Staubli VAL3: buildList.pgx

program buildList()
  local num l_nSize
  local string l_sEvent
  local num i
  local bool l_bFound
  local num l_nCount
  local string l_sEmpty
  local num j
begin
  call use:setSizeList(0,0,38,10)
  //call use:setSizeList(15,0,18,9)
  //建立对话款
  call use:listcreate("第1槽/6槽")
  //  for i=0 to 7
  //    call use:listadd(sMenu[i])
  //  endFor
 //   call use:selectNewField(nSelected,nIndex,nView)
  for i=0 to 7
    sTrsfNum[i,0]=toString("",data:pPoinTest[i].trsf.x)
    sTrsfNum[i,1]=toString("",data:pPoinTest[i].trsf.y)
    sTrsfNum[i,2]=toString("",data:pPoinTest[i].trsf.z)
    sTrsfNum[i,3]=toString("",data:pPoinTest[i].trsf.rx)
    sTrsfNum[i,4]=toString("",data:pPoinTest[i].trsf.ry)
    sTrsfNum[i,5]=toString("",data:pPoinTest[i].trsf.rz)
  endFor

  sWorkingmode[0]="0 安全过度点 Joint"
  sWorkingmode[1]="1 Appro(摆正点，{"+sTrsfNum[1,0]+","+sTrsfNum[1,1]+","+sTrsfNum[1,2]+","+sTrsfNum[1,3]+","+sTrsfNum[1,4]+","+sTrsfNum[1,5]+"})"
  sWorkingmode[2]="2 Appro(摆正点，{"+sTrsfNum[2,0]+","+sTrsfNum[2,1]+","+sTrsfNum[2,2]+","+sTrsfNum[2,3]+","+sTrsfNum[2,4]+","+sTrsfNum[2,5]+"})"
  sWorkingmode[3]="3 Appro(到位点，{"+sTrsfNum[3,0]+","+sTrsfNum[3,1]+","+sTrsfNum[3,2]+","+sTrsfNum[3,3]+","+sTrsfNum[3,4]+","+sTrsfNum[3,5]+"})"
  sWorkingmode[4]="4 Appro(到位点，{"+sTrsfNum[4,0]+","+sTrsfNum[4,1]+","+sTrsfNum[4,2]+","+sTrsfNum[4,3]+","+sTrsfNum[4,4]+","+sTrsfNum[4,5]+"})"
  sWorkingmode[5]="5 Appro(到位点，{"+sTrsfNum[5,0]+","+sTrsfNum[5,1]+","+sTrsfNum[5,2]+","+sTrsfNum[5,3]+","+sTrsfNum[5,4]+","+sTrsfNum[5,5]+"})"
  sWorkingmode[6]="6 Appro(摆正点，{"+sTrsfNum[6,0]+","+sTrsfNum[6,1]+","+sTrsfNum[6,2]+","+sTrsfNum[6,3]+","+sTrsfNum[6,4]+","+sTrsfNum[6,5]+"})"
  sWorkingmode[7]="7 Appro(摆正点，{"+sTrsfNum[7,0]+","+sTrsfNum[7,1]+","+sTrsfNum[7,2]+","+sTrsfNum[7,3]+","+sTrsfNum[7,4]+","+sTrsfNum[7,5]+"})"

  call use:listadd(sWorkingmode)
  call use:selectNewField(nSelected,nIndex,nView)
  call use:listupdate(0)
 // nIndex=data:nPage_Traj
 // call use:selectNewField(nSelected,nIndex,nView)
end
